Staubli VAL3: EllipsePoint.pgx

public program EllipsePoint(trsf& x_trSource[], trsf& x_trDest[], bool& x_bRes)
  local frame l_fFrame
  local num l_Dia
  local num l_nLegth
  local point l_pBuff
begin
  //腰形孔

  //根据三个trsf建立frame
  call SetFrame(x_trSource,l_fFrame,x_bRes)
  if !x_bRes
    return
  endIf
 link(l_fFrame,world)

  //圆弧的直径
  l_Dia=distance(x_trSource[1],x_trSource[2])
  l_nLegth=distance(x_trSource[0],x_trSource[1])



  link(l_pBuff,l_fFrame)
  l_pBuff.trsf={l_nLegth/2,0,0,0,0,0}
  x_trDest[0]=position(l_pBuff,world)

  l_pBuff.trsf={l_nLegth,0,0,0,0,0}
  x_trDest[1]=position(l_pBuff,world)

  l_pBuff.trsf={l_nLegth+l_Dia/2,l_Dia/2,0,0,0,0}
  x_trDest[2]=position(l_pBuff,world)

  l_pBuff.trsf={l_nLegth,l_Dia,0,0,0,0}
  x_trDest[3]=position(l_pBuff,world)

  l_pBuff.trsf={0,l_Dia,0,0,0,0}
  x_trDest[4]=position(l_pBuff,world)

  l_pBuff.trsf={-l_Dia/2,l_Dia/2,0,0,0,0}
  x_trDest[5]=position(l_pBuff,world)

  l_pBuff.trsf={0,0,0,0,0,0}
  x_trDest[6]=position(l_pBuff,world)

  x_trDest[7]=x_trDest[0]


    //圆心点
  l_pBuff.trsf={l_nLegth/2,min(l_nLegth/2,l_Dia/2),0,0,0,0}
  x_trDest[20]=position(l_pBuff,world)



  x_bRes=true

end
